(* Logix 5000 project; controller Hose_HP_Test_Rig_V1 vendor 1 type 14 code 149 rev 32.11; software revision 32.00; part 5 of 10 *)
(* tags used below, declared in another part *)
   CONS_ONS1 : BOOL;
   CONS_ONS2 : BOOL;
   CONS_ONS3 : BOOL;
   CONS_ONS4 : BOOL;
   DUMMY_VAL : REAL;
   EXHS_VAL_OFF_CE_STN1 : BOOL;
   EXHS_VAL_OFF_CE_STN2 : BOOL;
   EXHS_VAL_OFF_CE_STN3 : BOOL;
   FAULT_COMP_SENSOR : ALIAS FOR Local:2:I.Data.30;
   ONS42 : BOOL;
   ONS47 : BOOL;
   ONS48 : BOOL;
   ONS49 : BOOL;
   ONS53 : BOOL;
   ONS_74 : BOOL;
   ONS_75 : BOOL;
   ABORT_STN1 : BOOL;
   ABORT_STN2 : BOOL;
   ABORT_STN3 : BOOL;
   ABORT_STN4 : BOOL;
   AUTO_TEST_ON_STN1 : BOOL;
   AUTO_TEST_ON_STN2 : BOOL;
   AUTO_TEST_ON_STN3 : BOOL;
   AUTO_TEST_ON_STN4 : BOOL;
   BIN_MSG : DINT;
   BOTTOM_CLAMP_2BPR_HIGH : BOOL;
   BOTTOM_CLAMP_2BPR_LOW : BOOL;
   BOTTOM_CLAMP_4BPR_HIGH : BOOL;
   BOTTOM_CLAMP_4BPR_LOW : BOOL;
   BOTTOM_CLAMP_FAULT_STN1 : BOOL;
   BOTTOM_CLAMP_FAULT_STN2 : BOOL;
   BOTTOM_CLAMP_FAULT_STN3 : BOOL;
   BOTTOM_CLAMP_FAULT_STN4 : BOOL;
   BOTTOM_CLAMP_PR : REAL;
   BOTTOM_CLAMP_PR_DEL : TIMER;
   BOTTOM_CLAMP_PR_SEL : BOOL;
   BOTTOM_CLAMP_PR_SEQ : CLAMP_FAULT;
   BOTTOM_CLAMP_PS_STN2 : ALIAS FOR Local:2:I.Data.2;
   BOTTOM_CLAMP_PS_STN4 : ALIAS FOR Local:2:I.Data.12;
   BOTTOM_NOT_CLAMPED_STN1 : BOOL;
   CALB_START_PB_ONS_STN1 : BOOL;
   CALB_START_PB_ONS_STN2 : BOOL;
   CALB_START_PB_ONS_STN3 : BOOL;
   CALB_START_PB_ONS_STN4 : BOOL;
   CHECK_TRACE_STS_STN1 : BOOL;
   CLAMP_2BAR_HL : REAL;
   CLAMP_2BAR_LL : REAL;
   CLAMP_4BAR_HL : REAL;
   CLAMP_4BAR_LL : REAL;
   COMP_FAULT_STN1 : BOOL;
   CONS_CALB_ON_STN1 : BOOL;
   CONS_CALB_ON_STN2 : BOOL;
   CONS_CALB_ON_STN3 : BOOL;
   CONS_CALB_ON_STN4 : BOOL;
   CONS_CALB_TARRED_STN1 : BOOL;
   CONS_CALB_TARRED_STN2 : BOOL;
   CONS_CALB_TARRED_STN3 : BOOL;
   CONS_CALB_TARRED_STN4 : BOOL;
   CONS_DUMMIT_VAR : REAL;
   CONS_FILL_BLK_STN1 : CONSTRICTION_FILL_ON_SEQ;
   CONS_FILL_BLK_STN2 : CONSTRICTION_FILL_ON_SEQ;
   CONS_FILL_BLK_STN3 : CONSTRICTION_FILL_ON_SEQ;
   CONS_FILL_BLK_STN4 : CONSTRICTION_FILL_ON_SEQ;
   CONS_FILL_HIGH_STN1 : BOOL;
   CONS_FILL_HIGH_STN2 : BOOL;
   CONS_FILL_HIGH_STN3 : BOOL;
   CONS_FILL_HIGH_STN4 : BOOL;
   CONS_FILL_HL : REAL;
   CONS_FILL_LL : REAL;
   CONS_FILL_LOW_STN1 : BOOL;
   CONS_FILL_LOW_STN2 : BOOL;
   CONS_FILL_LOW_STN3 : BOOL;
   CONS_FILL_LOW_STN4 : BOOL;
   CONS_FILL_OFF_BLK_STN1 : CONSTRICTION_FILL_OFF_SEQ;
   CONS_FILL_OFF_BLK_STN2 : CONSTRICTION_FILL_OFF_SEQ;
   CONS_FILL_OFF_BLK_STN3 : CONSTRICTION_FILL_OFF_SEQ;
   CONS_FILL_OFF_BLK_STN4 : CONSTRICTION_FILL_OFF_SEQ;
   CONS_P2_STN1 : REAL;
   CONS_P2_STN2 : REAL;
   CONS_P2_STN3 : REAL;
   CONS_PR_BLK_STN1 : PR_CHECK;
   CONS_PR_BLK_STN2 : PR_CHECK;
   CONS_PR_BLK_STN3 : PR_CHECK;
   CONS_PR_BLK_STN4 : PR_CHECK;
   CONS_PR_P1_STN1 : REAL;
   CONS_PR_P1_STN2 : REAL;
   CONS_PR_P1_STN3 : REAL;
   CONS_PR_P1_STN4 : REAL;
   CONS_STS_STN1 : DINT;
   CONS_STS_STN2 : DINT;
   CONS_STS_STN3 : DINT;
   CONS_STS_STN4 : DINT;
   CONS_TEST_TIME_ACT : REAL;
   CONS_TEST_TIME_ACT_STN2 : REAL;
   CONS_TEST_TIME_ACT_STN3 : REAL;
   CONS_TEST_TIME_ACT_STN4 : REAL;
   CONS_TEST_TIME_SET : REAL;
   CONSTRICTION_BLK_STN1 : DROP_CHECK;
   CONSTRICTION_BLK_STN2 : DROP_CHECK;
   CONSTRICTION_BLK_STN3 : DROP_CHECK;
   CONSTRICTION_BLK_STN4 : DROP_CHECK;
   CONSTRICTION_FILL_OFF_STN1 : BOOL;
   CONSTRICTION_FILL_OFF_STN2 : BOOL;
   CONSTRICTION_FILL_OFF_STN3 : BOOL;
   CONSTRICTION_FILL_OFF_STN4 : BOOL;
   CONSTRICTION_FILL_VAL_STN1 : BOOL;
   CONSTRICTION_FILL_VAL_STN2 : BOOL;
   CONSTRICTION_FILL_VAL_STN3 : BOOL;
   CONSTRICTION_FILL_VAL_STN4 : BOOL;
   CONSTRICTION_NOK_STN1 : BOOL;
   CONSTRICTION_NOK_STN2 : BOOL;
   CONSTRICTION_NOK_STN3 : BOOL;
   CONSTRICTION_NOK_STN4 : BOOL;
   CONSTRICTION_OK_STN1 : BOOL;
   CONSTRICTION_OK_STN2 : BOOL;
   CONSTRICTION_OK_STN3 : BOOL;
   CONSTRICTION_OK_STN4 : BOOL;
   CONSTRICTION_TEST_ON_STN1 : BOOL;
   CONSTRICTION_TEST_ON_STN2 : BOOL;
   CONSTRICTION_TEST_ON_STN3 : BOOL;
   CONSTRICTION_TEST_ON_STN4 : BOOL;
   CYCLE_START_PB_STN1 : ALIAS FOR Local:1:I.Data.2;
   DOOR_CLOSE_ABORT_STN1 : BOOL;
   DOOR_NOT_CLOSED : BOOL;
   DOOR_NOT_OPEN_STN1 : BOOL;
   DROP_NOK_STN1 : BOOL;
   EC_STN1 : DINT;
   EC_STN2 : DINT;
   EC_STN3 : DINT;
   EC_STN4 : DINT;
   EMG_FAULT_CLR : BOOL;
   EMG_FAULTED_STN1 : BOOL;
   EMG_START_PB : ALIAS FOR Local:1:I.Data.6;
   EMG_STOP_PB_LH : ALIAS FOR Local:2:I.Data.23;
   EXHS_VAL_OFF_CE_STN4 : BOOL;
   EXHS_VAL_OFF_STN1 : BOOL;
   EXHS_VAL_OFF_STN2 : BOOL;
   EXHS_VAL_OFF_STN3 : BOOL;
   EXHS_VAL_OFF_STN4 : BOOL;
   EXHS_VAL_ON_STN1 : BOOL;
   EXHS_VAL_ON_STN2 : BOOL;
   EXHS_VAL_ON_STN3 : BOOL;
   EXHS_VAL_ON_STN4 : BOOL;
   FAIL_BIN_LOCK_PS : ALIAS FOR Local:2:I.Data.26;
   FAIL_CLR_ONS_STN1 : BOOL;
   FAIL_CLR_ONS_STN2 : BOOL;
   FAIL_CLR_ONS_STN3 : BOOL;
   FAIL_CLR_ONS_STN4 : BOOL;
   FAILED_STN1 : BOOL;
   FAILED_STN2 : BOOL;
   FAILED_STN3 : BOOL;
   FAULT_COUNT_STN1 : DINT;
   FAULT_COUNTER_STN1 : COUNTER;
   FAULTED_STN1 : BOOL;
   FAULTED_STN2 : BOOL;
   FAULTED_STN3 : BOOL;
   FAULTED_STN4 : BOOL;
   FILL_HIGH_STN1 : BOOL;
   FILL_LOW_STN1 : BOOL;
   FLT_CLR_ONS : BOOL;
   FLT_CLR_ONS_STN1 : BOOL;
   FLT_CLR_ONS_STN2 : BOOL;
   FLT_CLR_ONS_STN3 : BOOL;
   FLT_CLR_ONS_STN4 : BOOL;
   GOTO_FAULT_BIN_STN1 : DINT;
   HOME_COND_NOK_STN1 : BOOL;
   HOME_COND_OK_STN1 : BOOL;
   INIT_STN1 : BOOL;
   INIT_STN2 : BOOL;
   INIT_STN3 : BOOL;
   INIT_STN4 : BOOL;
   INLET_AIR_DPS : ALIAS FOR Local:1:I.Data.0;
   INLET_AIR_HPS : ALIAS FOR Local:1:I.Data.1;
   INLET_AIR_LOW : TIMER;
   INLET_AIR_SOL : ALIAS FOR Local:1:O.Data.0;
   LH_START_PB_STN2 : ALIAS FOR Local:1:I.Data.3;
   LH_START_PB_STN3 : ALIAS FOR Local:1:I.Data.4;
   LH_START_PB_STN4 : ALIAS FOR Local:1:I.Data.5;
   MSG_STN1 : DINT;
   MSG_STN2 : DINT;
   MSG_STN3 : DINT;
   MSG_STN4 : DINT;
   NO_COMP_FAULT_STN1 : BOOL;
   NO_SYSTEM_FAULT_STN1 : BOOL;
   NOT_FAILED_STN1 : BOOL;
   PASS_BIN_FULL : DINT;
   PR_DIFF_ACT_STN1 : REAL;
   PR_DIFF_ACT_STN2 : REAL;
   PR_DIFF_ACT_STN3 : REAL;
   PR_DIFF_ACT_STN4 : REAL;
   PR_DIFF_CALB_ACT : REAL;
   PR_DIFF_HL : REAL;
   PR_DIFF_LL : REAL;
   PR_DIFF_TARRED_STN1 : REAL;
   PR_DIFF_TARRED_STN2 : REAL;
   PR_DIFF_TARRED_STN3 : REAL;
   PR_DIFF_TARRED_STN4 : REAL;
   RETEST : BOOL;
   RST_DOOR_NOT_OPEN_STN1 : BOOL;
   RST_EXHS_VAL_OFF_STN1 : BOOL;
   RST_EXHS_VAL_OFF_STN2 : BOOL;
   RST_EXHS_VAL_OFF_STN3 : BOOL;
   RST_EXHS_VAL_OFF_STN4 : BOOL;
   RST_SEQ_ON_STN1 : BOOL;
   RST_SEQ_ON_STN2 : BOOL;
   RST_SEQ_ON_STN3 : BOOL;
   RST_SEQ_ON_STN4 : BOOL;
   SCR_STS : DINT[6];
   SEQ_NO_STN1 : DINT;
   SEQ_NO_STN2 : DINT;
   SEQ_NO_STN3 : DINT;
   SEQ_NO_STN4 : DINT;
   STAB_HIGH_STN1 : BOOL;
   STAB_LOW_STN1 : BOOL;
   STAMP_HL : REAL;
   STAMP_LL : REAL;
   STAMP_NOT_FWD : BOOL;
   STAMP_NOT_RET : BOOL;
   STAMP_PR : REAL;
   STAMP_PR_CHECK : TIMER;
   STAMP_PR_DEL : TIMER;
   STAMP_PR_HIGH_STN1 : BOOL;
   STAMP_PR_LOW_STN1 : BOOL;
   STAMP_SOL_STN1 : ALIAS FOR Local:1:O.Data.5;
   STS : DINT;
   SYSTEM_FAULT_STN1 : BOOL;
   TARRED_VALUE_STN1 : REAL;
   TARRED_VALUE_STN2 : REAL;
   TARRED_VALUE_STN3 : REAL;
   TARRED_VALUE_STN4 : REAL;
   TEST_ON_STN1 : BOOL;
   TEST_ON_STN2 : BOOL;
   TEST_ON_STN3 : BOOL;
   TEST_ON_STN4 : BOOL;
   TEST_STS_STN1 : DINT;
   TEST_STS_STN2 : DINT;
   TEST_STS_STN3 : DINT;
   TEST_STS_STN4 : DINT;
   TOP_CLAMP_2BPR_HIGH : BOOL;
   TOP_CLAMP_2BPR_LOW : BOOL;
   TOP_CLAMP_4BPR_HIGH : BOOL;
   TOP_CLAMP_4BPR_LOW : BOOL;
   TOP_CLAMP_FAULT_STN1 : BOOL;
   TOP_CLAMP_FAULT_STN2 : BOOL;
   TOP_CLAMP_FAULT_STN3 : BOOL;
   TOP_CLAMP_FAULT_STN4 : BOOL;
   TOP_CLAMP_PR : REAL;
   TOP_CLAMP_PR_CHK_STN1 : TIMER;
   TOP_CLAMP_PR_DEL : TIMER;
   TOP_CLAMP_PR_SEL : BOOL;
(* MainProgram, continued *)

ROUTINE Constriction_Stn1   (* ladder *)
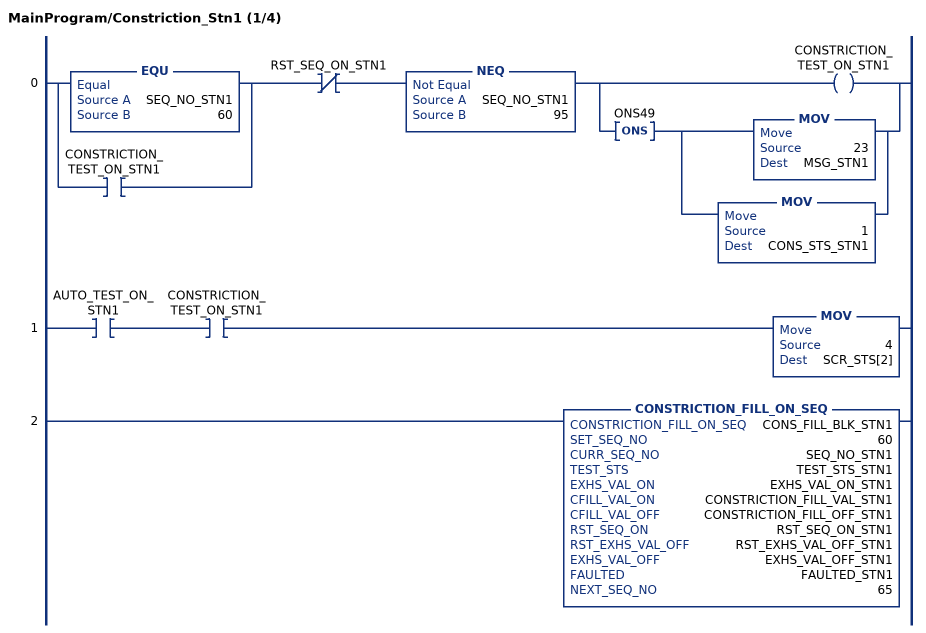
   0: [EQU(SEQ_NO_STN1,60) ,XIC(CONSTRICTION_TEST_ON_STN1) ]XIO(RST_SEQ_ON_STN1)NEQ(SEQ_NO_STN1,95)[OTE(CONSTRICTION_TEST_ON_STN1) ,ONS(ONS49) [MOV(23,MSG_STN1) ,MOV(1,CONS_STS_STN1) ] ];
   1: XIC(AUTO_TEST_ON_STN1)XIC(CONSTRICTION_TEST_ON_STN1)MOV(4,SCR_STS[2]);
   2: CONSTRICTION_FILL_ON_SEQ(CONS_FILL_BLK_STN1,60,SEQ_NO_STN1,TEST_STS_STN1,EXHS_VAL_ON_STN1,CONSTRICTION_FILL_VAL_STN1,CONSTRICTION_FILL_OFF_STN1,RST_SEQ_ON_STN1,RST_EXHS_VAL_OFF_STN1,EXHS_VAL_OFF_STN1,FAULTED_STN1,65);
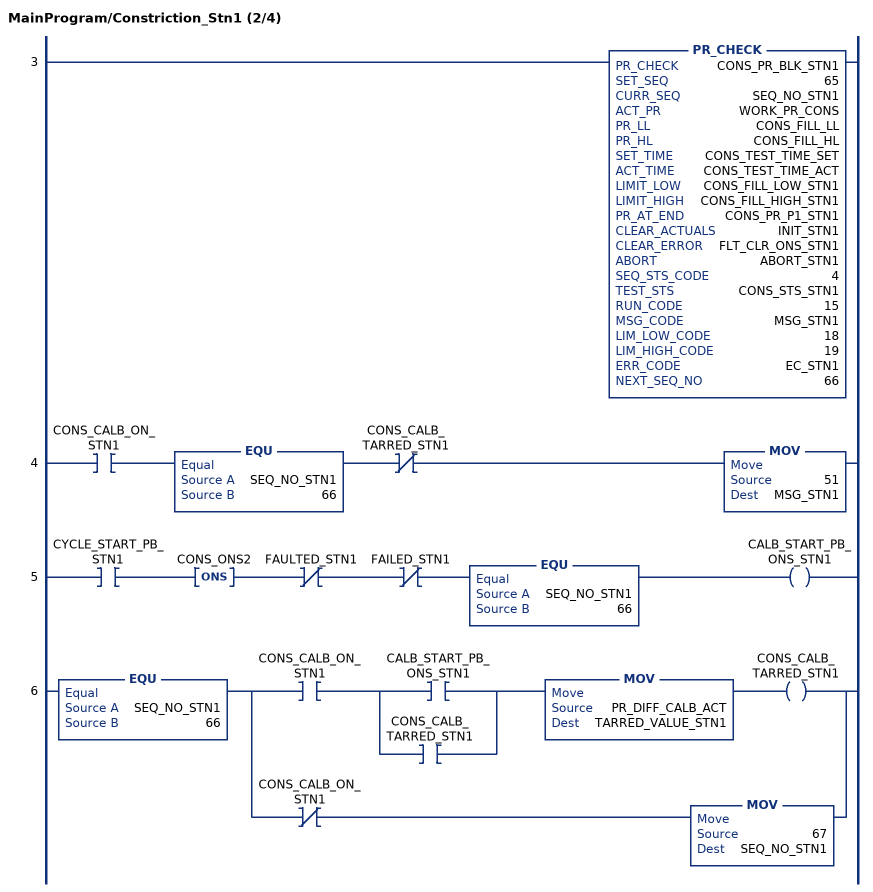
   3: PR_CHECK(CONS_PR_BLK_STN1,65,SEQ_NO_STN1,WORK_PR_CONS,CONS_FILL_LL,CONS_FILL_HL,CONS_TEST_TIME_SET,CONS_TEST_TIME_ACT,CONS_FILL_LOW_STN1,CONS_FILL_HIGH_STN1,CONS_PR_P1_STN1,INIT_STN1,FLT_CLR_ONS_STN1,ABORT_STN1,4,CONS_STS_STN1,15,MSG_STN1,18,19,EC_STN1,66);
   4: XIC(CONS_CALB_ON_STN1)EQU(SEQ_NO_STN1,66)XIO(CONS_CALB_TARRED_STN1)MOV(51,MSG_STN1);
   5: XIC(CYCLE_START_PB_STN1)ONS(CONS_ONS2)XIO(FAULTED_STN1)XIO(FAILED_STN1)EQU(SEQ_NO_STN1,66)OTE(CALB_START_PB_ONS_STN1);
   6: EQU(SEQ_NO_STN1,66)[XIC(CONS_CALB_ON_STN1) [XIC(CALB_START_PB_ONS_STN1) ,XIC(CONS_CALB_TARRED_STN1) ] MOV(PR_DIFF_CALB_ACT,TARRED_VALUE_STN1) OTE(CONS_CALB_TARRED_STN1) ,XIO(CONS_CALB_ON_STN1) MOV(67,SEQ_NO_STN1) ];
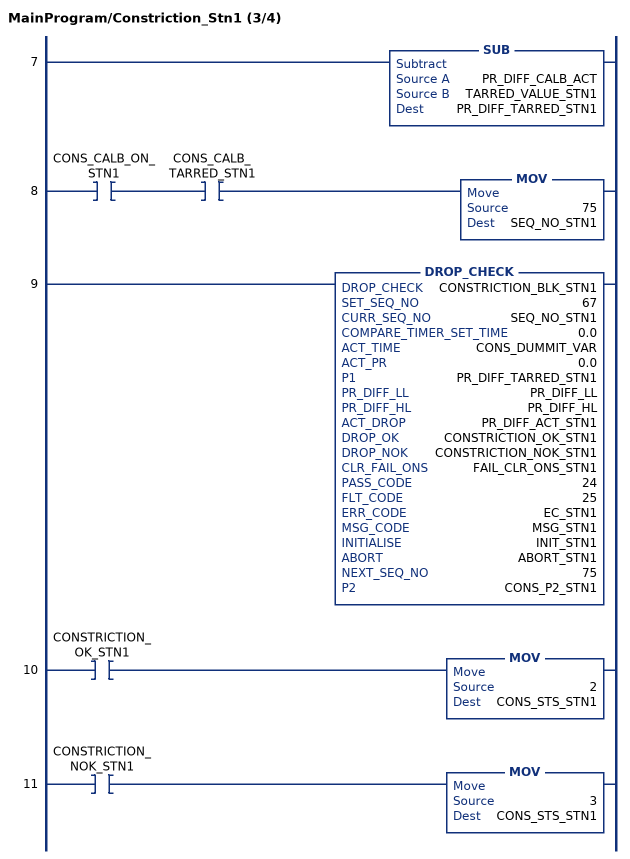
   7: SUB(PR_DIFF_CALB_ACT,TARRED_VALUE_STN1,PR_DIFF_TARRED_STN1);
   8: XIC(CONS_CALB_ON_STN1)XIC(CONS_CALB_TARRED_STN1)MOV(75,SEQ_NO_STN1);
   9: DROP_CHECK(CONSTRICTION_BLK_STN1,67,SEQ_NO_STN1,0.0,CONS_DUMMIT_VAR,0.0,PR_DIFF_TARRED_STN1,PR_DIFF_LL,PR_DIFF_HL,PR_DIFF_ACT_STN1,CONSTRICTION_OK_STN1,CONSTRICTION_NOK_STN1,FAIL_CLR_ONS_STN1,24,25,EC_STN1,MSG_STN1,INIT_STN1,ABORT_STN1,75,CONS_P2_STN1);
   10: XIC(CONSTRICTION_OK_STN1)MOV(2,CONS_STS_STN1);
   11: XIC(CONSTRICTION_NOK_STN1)MOV(3,CONS_STS_STN1);
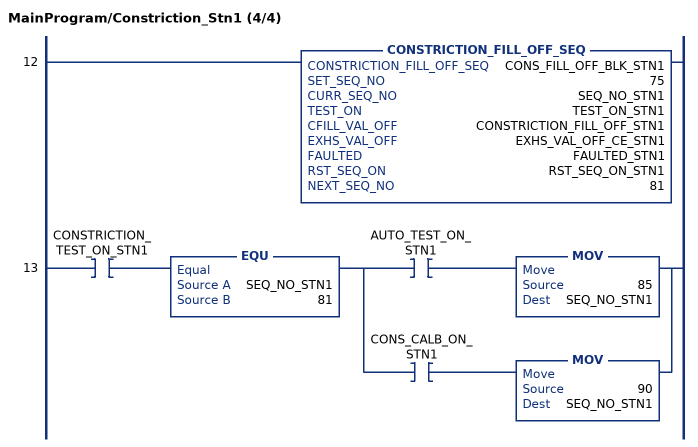
   12: CONSTRICTION_FILL_OFF_SEQ(CONS_FILL_OFF_BLK_STN1,75,SEQ_NO_STN1,TEST_ON_STN1,CONSTRICTION_FILL_OFF_STN1,EXHS_VAL_OFF_CE_STN1,FAULTED_STN1,RST_SEQ_ON_STN1,81);
   13: XIC(CONSTRICTION_TEST_ON_STN1)EQU(SEQ_NO_STN1,81)[XIC(AUTO_TEST_ON_STN1) MOV(85,SEQ_NO_STN1) ,XIC(CONS_CALB_ON_STN1) MOV(90,SEQ_NO_STN1) ];
END_ROUTINE

ROUTINE Constriction_Stn2   (* ladder *)
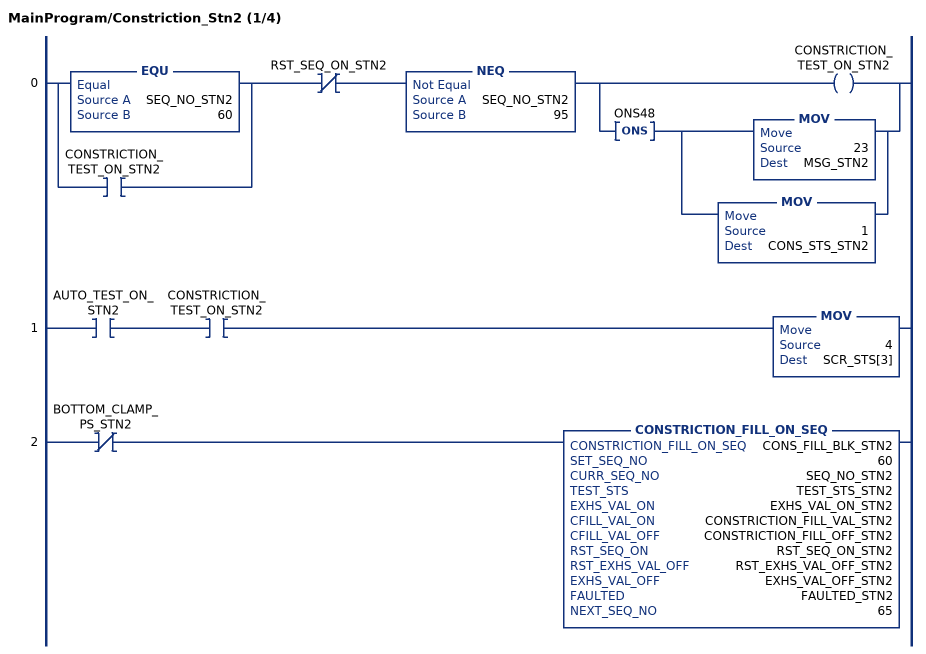
   0: [EQU(SEQ_NO_STN2,60) ,XIC(CONSTRICTION_TEST_ON_STN2) ]XIO(RST_SEQ_ON_STN2)NEQ(SEQ_NO_STN2,95)[OTE(CONSTRICTION_TEST_ON_STN2) ,ONS(ONS48) [MOV(23,MSG_STN2) ,MOV(1,CONS_STS_STN2) ] ];
   1: XIC(AUTO_TEST_ON_STN2)XIC(CONSTRICTION_TEST_ON_STN2)MOV(4,SCR_STS[3]);
   2: XIO(BOTTOM_CLAMP_PS_STN2)CONSTRICTION_FILL_ON_SEQ(CONS_FILL_BLK_STN2,60,SEQ_NO_STN2,TEST_STS_STN2,EXHS_VAL_ON_STN2,CONSTRICTION_FILL_VAL_STN2,CONSTRICTION_FILL_OFF_STN2,RST_SEQ_ON_STN2,RST_EXHS_VAL_OFF_STN2,EXHS_VAL_OFF_STN2,FAULTED_STN2,65);
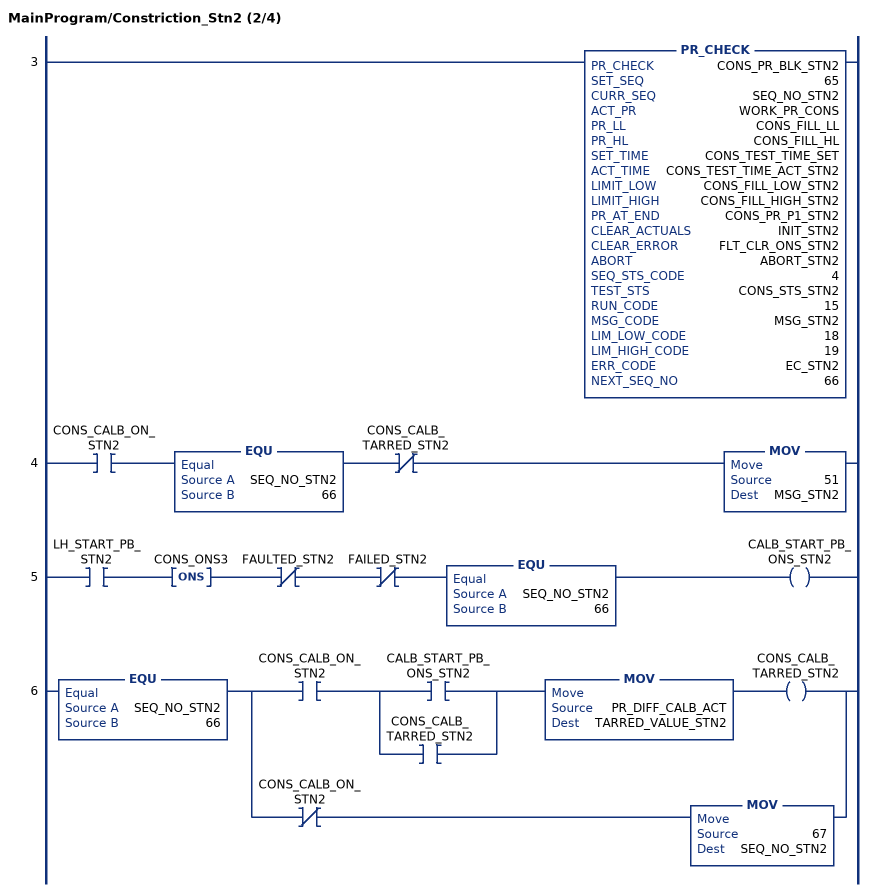
   3: PR_CHECK(CONS_PR_BLK_STN2,65,SEQ_NO_STN2,WORK_PR_CONS,CONS_FILL_LL,CONS_FILL_HL,CONS_TEST_TIME_SET,CONS_TEST_TIME_ACT_STN2,CONS_FILL_LOW_STN2,CONS_FILL_HIGH_STN2,CONS_PR_P1_STN2,INIT_STN2,FLT_CLR_ONS_STN2,ABORT_STN2,4,CONS_STS_STN2,15,MSG_STN2,18,19,EC_STN2,66);
   4: XIC(CONS_CALB_ON_STN2)EQU(SEQ_NO_STN2,66)XIO(CONS_CALB_TARRED_STN2)MOV(51,MSG_STN2);
   5: XIC(LH_START_PB_STN2)ONS(CONS_ONS3)XIO(FAULTED_STN2)XIO(FAILED_STN2)EQU(SEQ_NO_STN2,66)OTE(CALB_START_PB_ONS_STN2);
   6: EQU(SEQ_NO_STN2,66)[XIC(CONS_CALB_ON_STN2) [XIC(CALB_START_PB_ONS_STN2) ,XIC(CONS_CALB_TARRED_STN2) ] MOV(PR_DIFF_CALB_ACT,TARRED_VALUE_STN2) OTE(CONS_CALB_TARRED_STN2) ,XIO(CONS_CALB_ON_STN2) MOV(67,SEQ_NO_STN2) ];
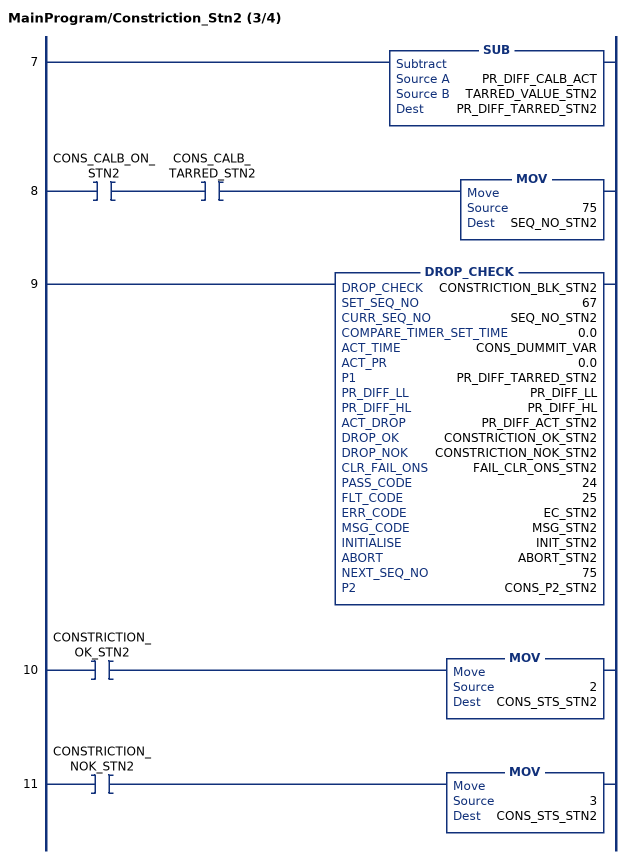
   7: SUB(PR_DIFF_CALB_ACT,TARRED_VALUE_STN2,PR_DIFF_TARRED_STN2);
   8: XIC(CONS_CALB_ON_STN2)XIC(CONS_CALB_TARRED_STN2)MOV(75,SEQ_NO_STN2);
   9: DROP_CHECK(CONSTRICTION_BLK_STN2,67,SEQ_NO_STN2,0.0,CONS_DUMMIT_VAR,0.0,PR_DIFF_TARRED_STN2,PR_DIFF_LL,PR_DIFF_HL,PR_DIFF_ACT_STN2,CONSTRICTION_OK_STN2,CONSTRICTION_NOK_STN2,FAIL_CLR_ONS_STN2,24,25,EC_STN2,MSG_STN2,INIT_STN2,ABORT_STN2,75,CONS_P2_STN2);
   10: XIC(CONSTRICTION_OK_STN2)MOV(2,CONS_STS_STN2);
   11: XIC(CONSTRICTION_NOK_STN2)MOV(3,CONS_STS_STN2);
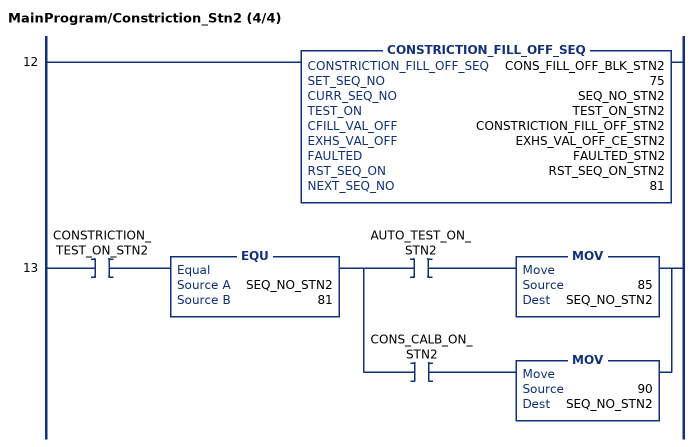
   12: CONSTRICTION_FILL_OFF_SEQ(CONS_FILL_OFF_BLK_STN2,75,SEQ_NO_STN2,TEST_ON_STN2,CONSTRICTION_FILL_OFF_STN2,EXHS_VAL_OFF_CE_STN2,FAULTED_STN2,RST_SEQ_ON_STN2,81);
   13: XIC(CONSTRICTION_TEST_ON_STN2)EQU(SEQ_NO_STN2,81)[XIC(AUTO_TEST_ON_STN2) MOV(85,SEQ_NO_STN2) ,XIC(CONS_CALB_ON_STN2) MOV(90,SEQ_NO_STN2) ];
END_ROUTINE

ROUTINE Constriction_Stn3   (* ladder *)
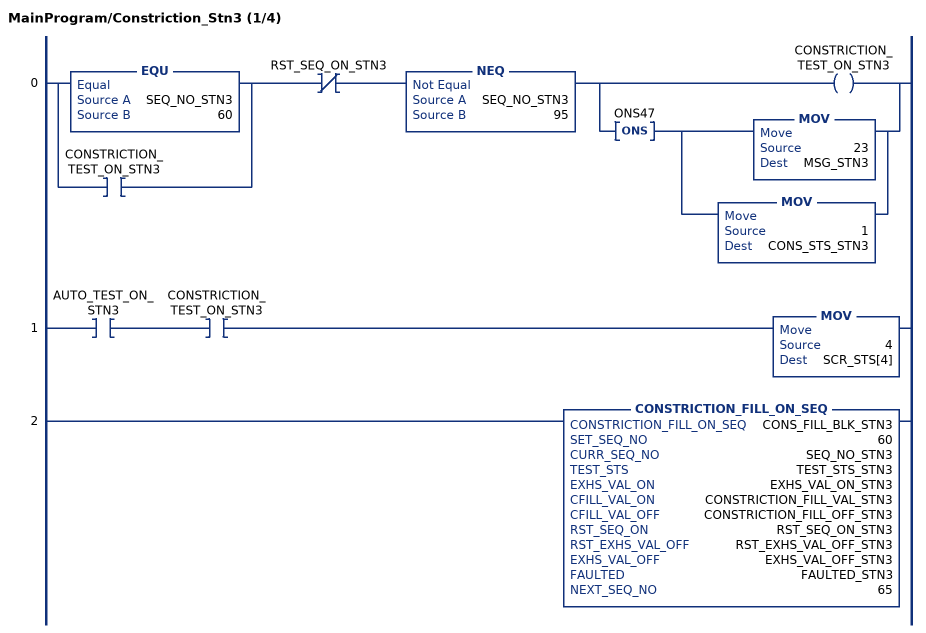
   0: [EQU(SEQ_NO_STN3,60) ,XIC(CONSTRICTION_TEST_ON_STN3) ]XIO(RST_SEQ_ON_STN3)NEQ(SEQ_NO_STN3,95)[OTE(CONSTRICTION_TEST_ON_STN3) ,ONS(ONS47) [MOV(23,MSG_STN3) ,MOV(1,CONS_STS_STN3) ] ];
   1: XIC(AUTO_TEST_ON_STN3)XIC(CONSTRICTION_TEST_ON_STN3)MOV(4,SCR_STS[4]);
   2: CONSTRICTION_FILL_ON_SEQ(CONS_FILL_BLK_STN3,60,SEQ_NO_STN3,TEST_STS_STN3,EXHS_VAL_ON_STN3,CONSTRICTION_FILL_VAL_STN3,CONSTRICTION_FILL_OFF_STN3,RST_SEQ_ON_STN3,RST_EXHS_VAL_OFF_STN3,EXHS_VAL_OFF_STN3,FAULTED_STN3,65);
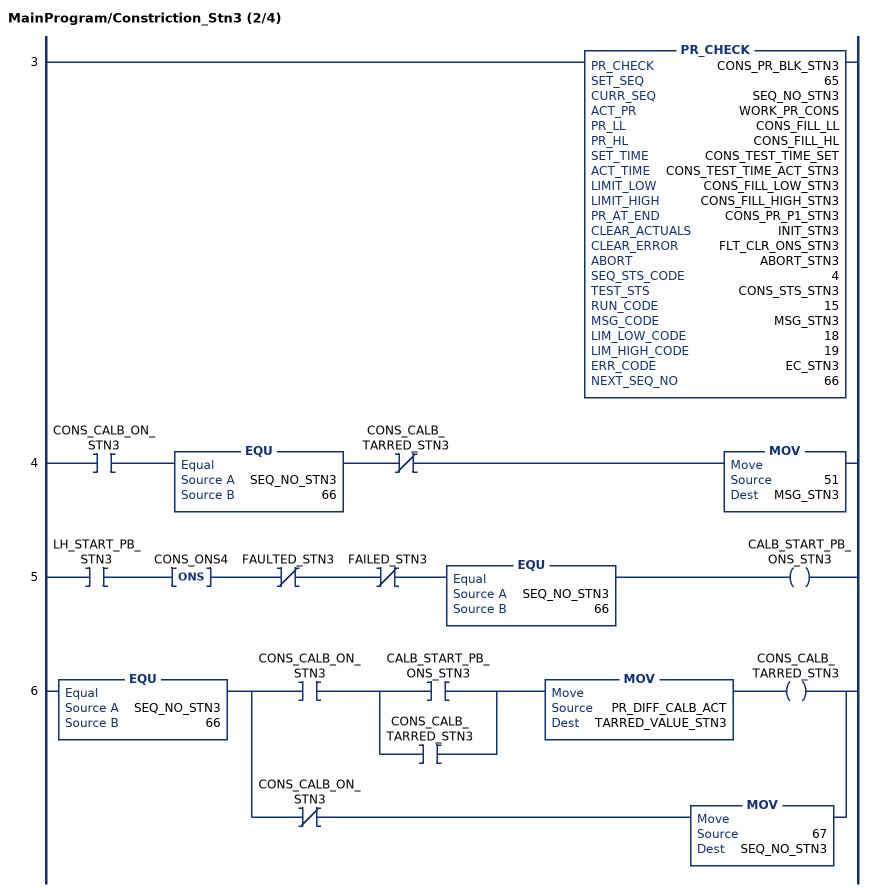
   3: PR_CHECK(CONS_PR_BLK_STN3,65,SEQ_NO_STN3,WORK_PR_CONS,CONS_FILL_LL,CONS_FILL_HL,CONS_TEST_TIME_SET,CONS_TEST_TIME_ACT_STN3,CONS_FILL_LOW_STN3,CONS_FILL_HIGH_STN3,CONS_PR_P1_STN3,INIT_STN3,FLT_CLR_ONS_STN3,ABORT_STN3,4,CONS_STS_STN3,15,MSG_STN3,18,19,EC_STN3,66);
   4: XIC(CONS_CALB_ON_STN3)EQU(SEQ_NO_STN3,66)XIO(CONS_CALB_TARRED_STN3)MOV(51,MSG_STN3);
   5: XIC(LH_START_PB_STN3)ONS(CONS_ONS4)XIO(FAULTED_STN3)XIO(FAILED_STN3)EQU(SEQ_NO_STN3,66)OTE(CALB_START_PB_ONS_STN3);
   6: EQU(SEQ_NO_STN3,66)[XIC(CONS_CALB_ON_STN3) [XIC(CALB_START_PB_ONS_STN3) ,XIC(CONS_CALB_TARRED_STN3) ] MOV(PR_DIFF_CALB_ACT,TARRED_VALUE_STN3) OTE(CONS_CALB_TARRED_STN3) ,XIO(CONS_CALB_ON_STN3) MOV(67,SEQ_NO_STN3) ];
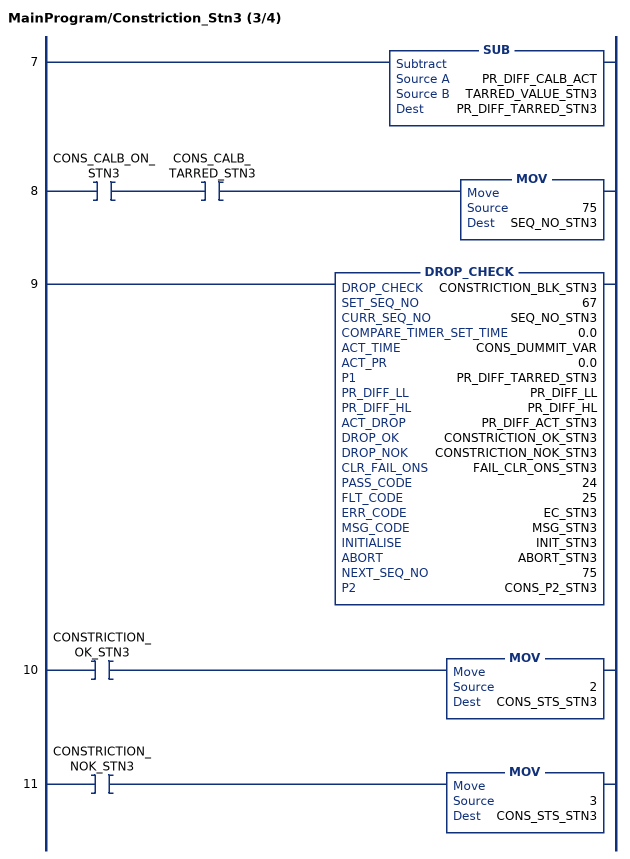
   7: SUB(PR_DIFF_CALB_ACT,TARRED_VALUE_STN3,PR_DIFF_TARRED_STN3);
   8: XIC(CONS_CALB_ON_STN3)XIC(CONS_CALB_TARRED_STN3)MOV(75,SEQ_NO_STN3);
   9: DROP_CHECK(CONSTRICTION_BLK_STN3,67,SEQ_NO_STN3,0.0,CONS_DUMMIT_VAR,0.0,PR_DIFF_TARRED_STN3,PR_DIFF_LL,PR_DIFF_HL,PR_DIFF_ACT_STN3,CONSTRICTION_OK_STN3,CONSTRICTION_NOK_STN3,FAIL_CLR_ONS_STN3,24,25,EC_STN3,MSG_STN3,INIT_STN3,ABORT_STN3,75,CONS_P2_STN3);
   10: XIC(CONSTRICTION_OK_STN3)MOV(2,CONS_STS_STN3);
   11: XIC(CONSTRICTION_NOK_STN3)MOV(3,CONS_STS_STN3);
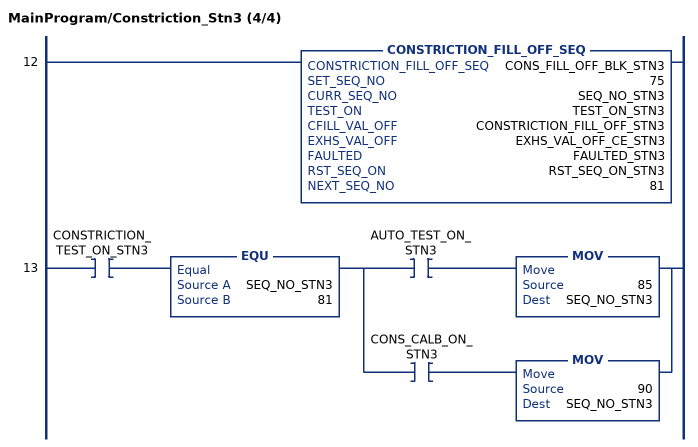
   12: CONSTRICTION_FILL_OFF_SEQ(CONS_FILL_OFF_BLK_STN3,75,SEQ_NO_STN3,TEST_ON_STN3,CONSTRICTION_FILL_OFF_STN3,EXHS_VAL_OFF_CE_STN3,FAULTED_STN3,RST_SEQ_ON_STN3,81);
   13: XIC(CONSTRICTION_TEST_ON_STN3)EQU(SEQ_NO_STN3,81)[XIC(AUTO_TEST_ON_STN3) MOV(85,SEQ_NO_STN3) ,XIC(CONS_CALB_ON_STN3) MOV(90,SEQ_NO_STN3) ];
END_ROUTINE

ROUTINE Constriction_Stn4   (* ladder *)
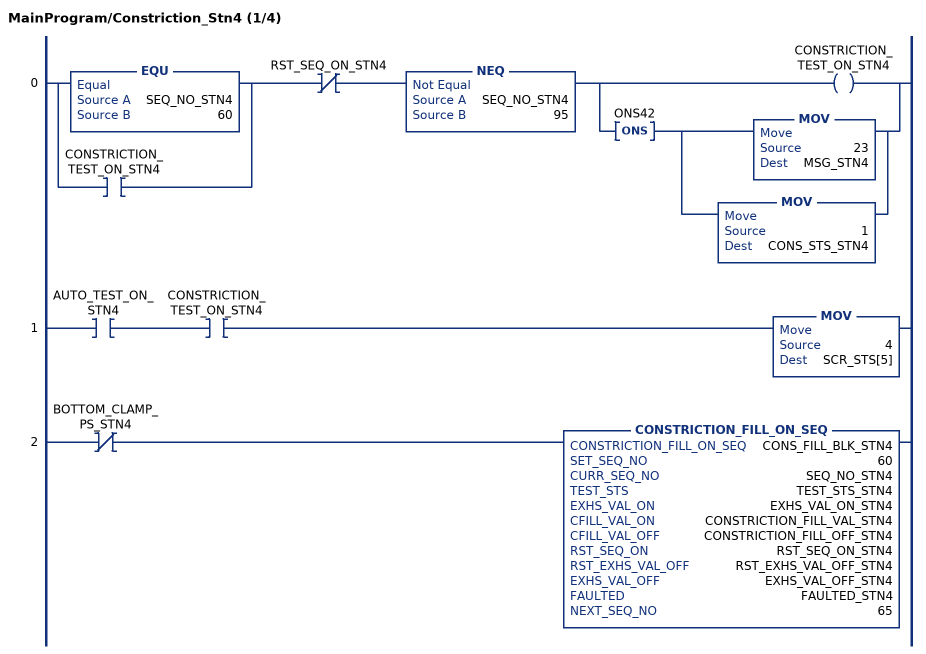
   0: [EQU(SEQ_NO_STN4,60) ,XIC(CONSTRICTION_TEST_ON_STN4) ]XIO(RST_SEQ_ON_STN4)NEQ(SEQ_NO_STN4,95)[OTE(CONSTRICTION_TEST_ON_STN4) ,ONS(ONS42) [MOV(23,MSG_STN4) ,MOV(1,CONS_STS_STN4) ] ];
   1: XIC(AUTO_TEST_ON_STN4)XIC(CONSTRICTION_TEST_ON_STN4)MOV(4,SCR_STS[5]);
   2: XIO(BOTTOM_CLAMP_PS_STN4)CONSTRICTION_FILL_ON_SEQ(CONS_FILL_BLK_STN4,60,SEQ_NO_STN4,TEST_STS_STN4,EXHS_VAL_ON_STN4,CONSTRICTION_FILL_VAL_STN4,CONSTRICTION_FILL_OFF_STN4,RST_SEQ_ON_STN4,RST_EXHS_VAL_OFF_STN4,EXHS_VAL_OFF_STN4,FAULTED_STN4,65);
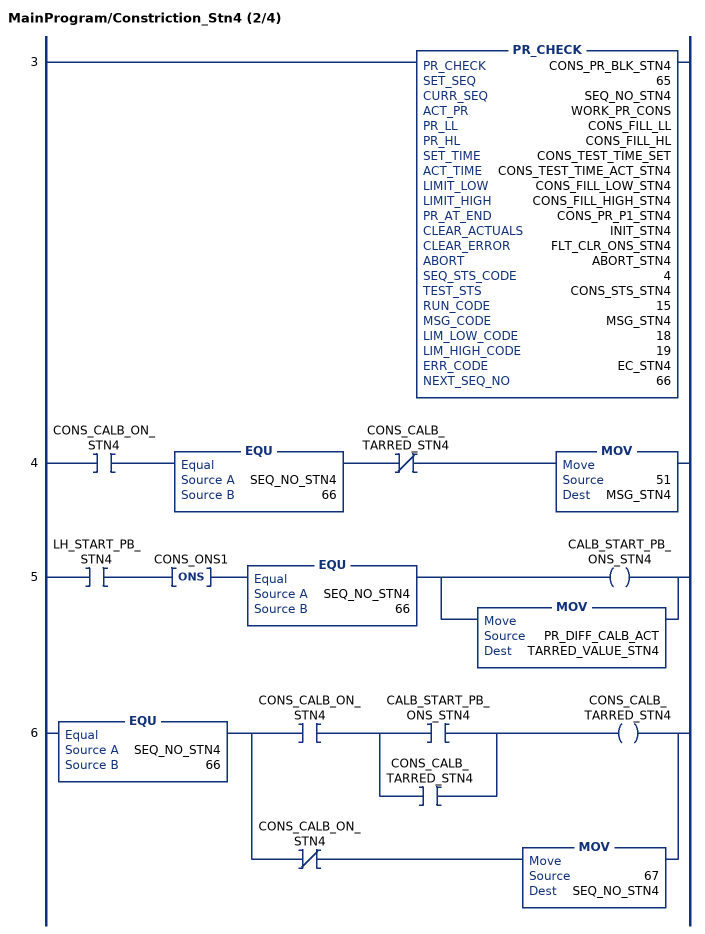
   3: PR_CHECK(CONS_PR_BLK_STN4,65,SEQ_NO_STN4,WORK_PR_CONS,CONS_FILL_LL,CONS_FILL_HL,CONS_TEST_TIME_SET,CONS_TEST_TIME_ACT_STN4,CONS_FILL_LOW_STN4,CONS_FILL_HIGH_STN4,CONS_PR_P1_STN4,INIT_STN4,FLT_CLR_ONS_STN4,ABORT_STN4,4,CONS_STS_STN4,15,MSG_STN4,18,19,EC_STN4,66);
   4: XIC(CONS_CALB_ON_STN4)EQU(SEQ_NO_STN4,66)XIO(CONS_CALB_TARRED_STN4)MOV(51,MSG_STN4);
   5: XIC(LH_START_PB_STN4)ONS(CONS_ONS1)EQU(SEQ_NO_STN4,66)[OTE(CALB_START_PB_ONS_STN4) ,MOV(PR_DIFF_CALB_ACT,TARRED_VALUE_STN4) ];
   6: EQU(SEQ_NO_STN4,66)[XIC(CONS_CALB_ON_STN4) [XIC(CALB_START_PB_ONS_STN4) ,XIC(CONS_CALB_TARRED_STN4) ] OTE(CONS_CALB_TARRED_STN4) ,XIO(CONS_CALB_ON_STN4) MOV(67,SEQ_NO_STN4) ];
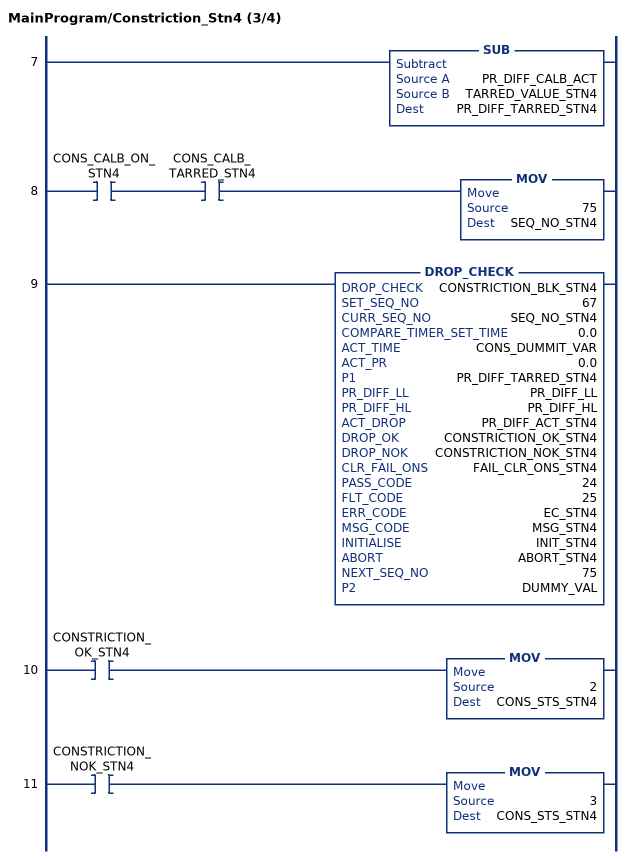
   7: SUB(PR_DIFF_CALB_ACT,TARRED_VALUE_STN4,PR_DIFF_TARRED_STN4);
   8: XIC(CONS_CALB_ON_STN4)XIC(CONS_CALB_TARRED_STN4)MOV(75,SEQ_NO_STN4);
   9: DROP_CHECK(CONSTRICTION_BLK_STN4,67,SEQ_NO_STN4,0.0,CONS_DUMMIT_VAR,0.0,PR_DIFF_TARRED_STN4,PR_DIFF_LL,PR_DIFF_HL,PR_DIFF_ACT_STN4,CONSTRICTION_OK_STN4,CONSTRICTION_NOK_STN4,FAIL_CLR_ONS_STN4,24,25,EC_STN4,MSG_STN4,INIT_STN4,ABORT_STN4,75,DUMMY_VAL);
   10: XIC(CONSTRICTION_OK_STN4)MOV(2,CONS_STS_STN4);
   11: XIC(CONSTRICTION_NOK_STN4)MOV(3,CONS_STS_STN4);
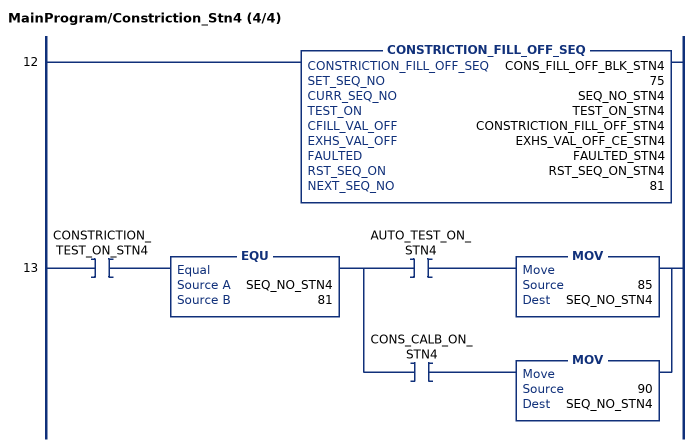
   12: CONSTRICTION_FILL_OFF_SEQ(CONS_FILL_OFF_BLK_STN4,75,SEQ_NO_STN4,TEST_ON_STN4,CONSTRICTION_FILL_OFF_STN4,EXHS_VAL_OFF_CE_STN4,FAULTED_STN4,RST_SEQ_ON_STN4,81);
   13: XIC(CONSTRICTION_TEST_ON_STN4)EQU(SEQ_NO_STN4,81)[XIC(AUTO_TEST_ON_STN4) MOV(85,SEQ_NO_STN4) ,XIC(CONS_CALB_ON_STN4) MOV(90,SEQ_NO_STN4) ];
END_ROUTINE

ROUTINE Fault_Fail_Msg   (* ladder *)
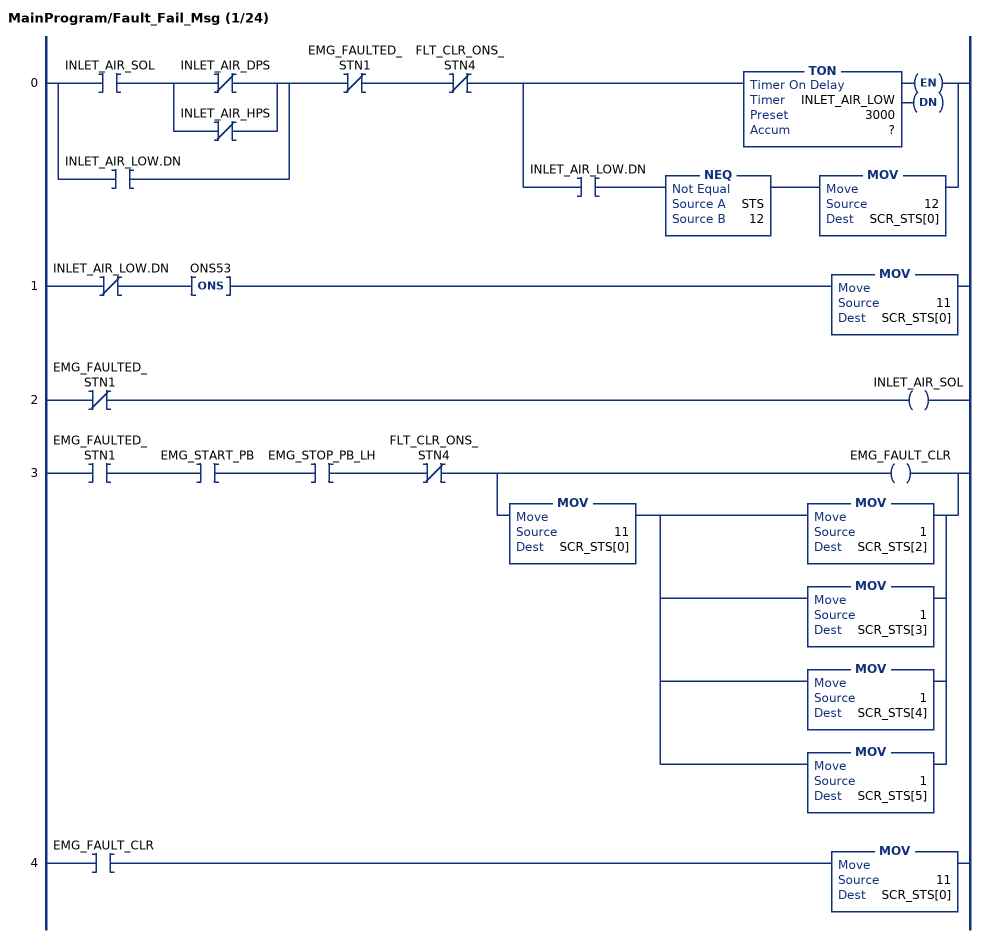
   0: [XIC(INLET_AIR_SOL) [XIO(INLET_AIR_DPS) ,XIO(INLET_AIR_HPS) ] ,XIC(INLET_AIR_LOW.DN) ]XIO(EMG_FAULTED_STN1)XIO(FLT_CLR_ONS_STN4)[TON(INLET_AIR_LOW,?,?) ,XIC(INLET_AIR_LOW.DN) NEQ(STS,12) MOV(12,SCR_STS[0]) ];
   1: XIO(INLET_AIR_LOW.DN)ONS(ONS53)MOV(11,SCR_STS[0]);
   2: XIO(EMG_FAULTED_STN1)OTE(INLET_AIR_SOL);
   3: XIC(EMG_FAULTED_STN1)XIC(EMG_START_PB)XIC(EMG_STOP_PB_LH)XIO(FLT_CLR_ONS_STN4)[OTE(EMG_FAULT_CLR) ,MOV(11,SCR_STS[0]) [MOV(1,SCR_STS[2]) ,MOV(1,SCR_STS[3]) ,MOV(1,SCR_STS[4]) ,MOV(1,SCR_STS[5]) ] ];
   4: XIC(EMG_FAULT_CLR)MOV(11,SCR_STS[0]);
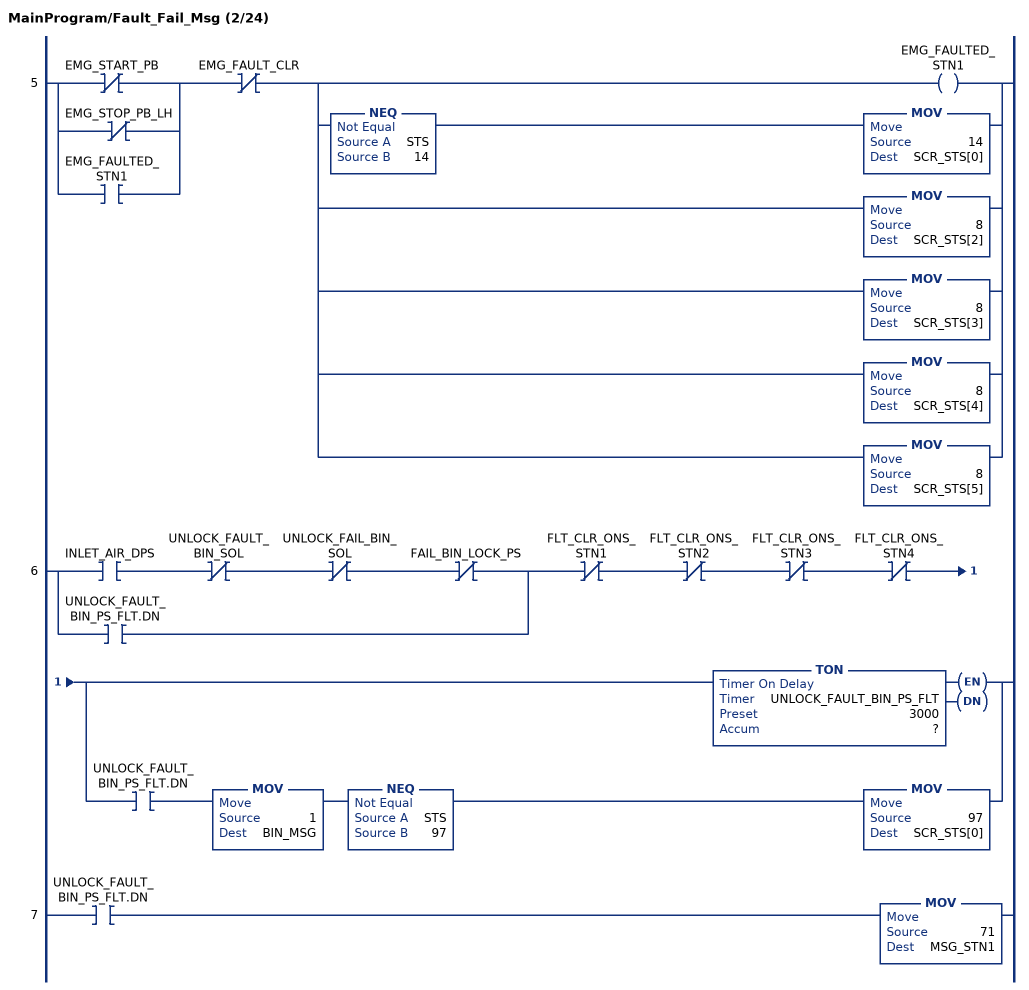
   5: [XIO(EMG_START_PB) ,XIO(EMG_STOP_PB_LH) ,XIC(EMG_FAULTED_STN1) ]XIO(EMG_FAULT_CLR)[OTE(EMG_FAULTED_STN1) ,NEQ(STS,14) MOV(14,SCR_STS[0]) ,MOV(8,SCR_STS[2]) ,MOV(8,SCR_STS[3]) ,MOV(8,SCR_STS[4]) ,MOV(8,SCR_STS[5]) ];
   6: [XIC(INLET_AIR_DPS) XIO(UNLOCK_FAULT_BIN_SOL) XIO(UNLOCK_FAIL_BIN_SOL) XIO(FAIL_BIN_LOCK_PS) ,XIC(UNLOCK_FAULT_BIN_PS_FLT.DN) ]XIO(FLT_CLR_ONS_STN1)XIO(FLT_CLR_ONS_STN2)XIO(FLT_CLR_ONS_STN3)XIO(FLT_CLR_ONS_STN4)[TON(UNLOCK_FAULT_BIN_PS_FLT,?,?) ,XIC(UNLOCK_FAULT_BIN_PS_FLT.DN) MOV(1,BIN_MSG) NEQ(STS,97) MOV(97,SCR_STS[0]) ];
   7: XIC(UNLOCK_FAULT_BIN_PS_FLT.DN)MOV(71,MSG_STN1);
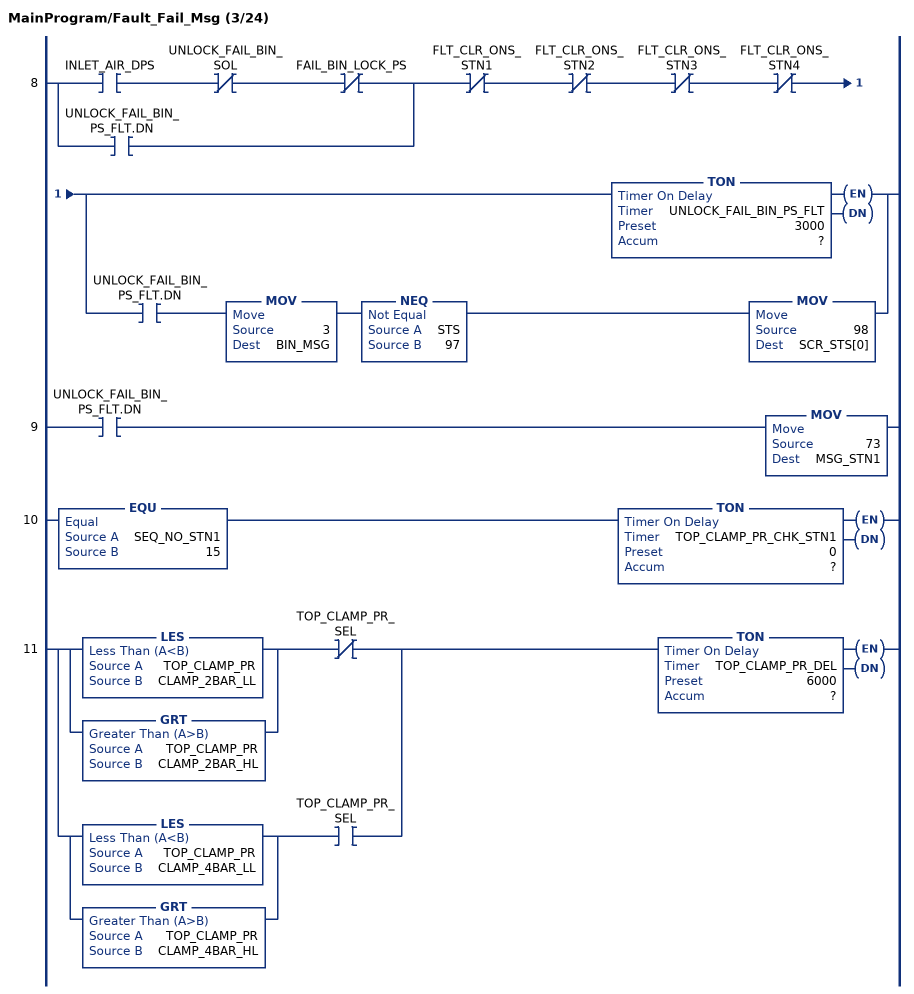
   8: [XIC(INLET_AIR_DPS) XIO(UNLOCK_FAIL_BIN_SOL) XIO(FAIL_BIN_LOCK_PS) ,XIC(UNLOCK_FAIL_BIN_PS_FLT.DN) ]XIO(FLT_CLR_ONS_STN1)XIO(FLT_CLR_ONS_STN2)XIO(FLT_CLR_ONS_STN3)XIO(FLT_CLR_ONS_STN4)[TON(UNLOCK_FAIL_BIN_PS_FLT,?,?) ,XIC(UNLOCK_FAIL_BIN_PS_FLT.DN) MOV(3,BIN_MSG) NEQ(STS,97) MOV(98,SCR_STS[0]) ];
   9: XIC(UNLOCK_FAIL_BIN_PS_FLT.DN)MOV(73,MSG_STN1);
   10: EQU(SEQ_NO_STN1,15)TON(TOP_CLAMP_PR_CHK_STN1,?,?);
   11: [[LES(TOP_CLAMP_PR,CLAMP_2BAR_LL) ,GRT(TOP_CLAMP_PR,CLAMP_2BAR_HL) ] XIO(TOP_CLAMP_PR_SEL) ,[LES(TOP_CLAMP_PR,CLAMP_4BAR_LL) ,GRT(TOP_CLAMP_PR,CLAMP_4BAR_HL) ] XIC(TOP_CLAMP_PR_SEL) ]TON(TOP_CLAMP_PR_DEL,?,?);
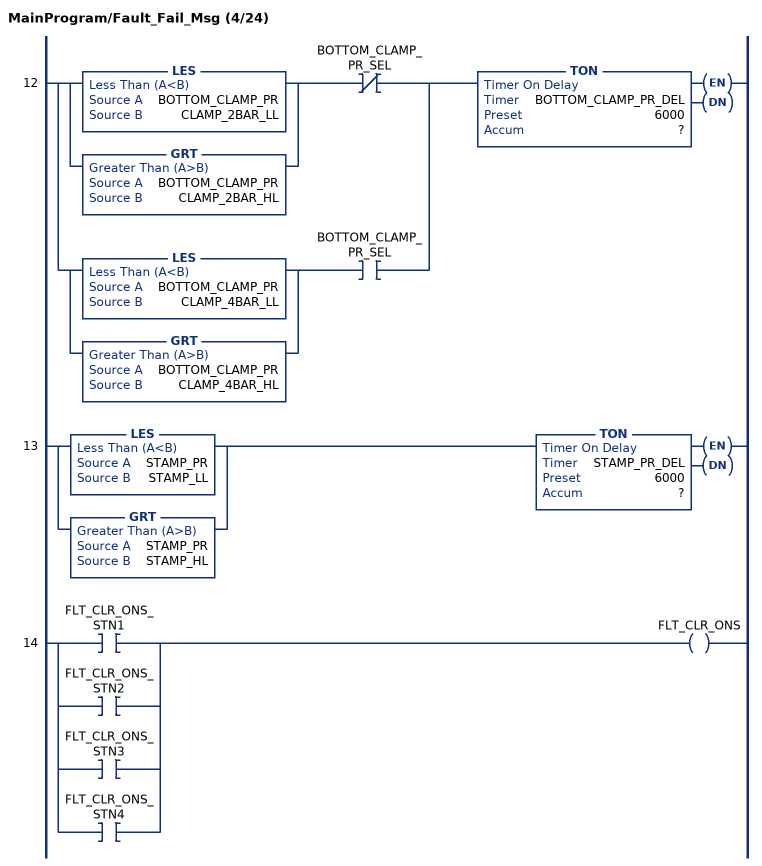
   12: [[LES(BOTTOM_CLAMP_PR,CLAMP_2BAR_LL) ,GRT(BOTTOM_CLAMP_PR,CLAMP_2BAR_HL) ] XIO(BOTTOM_CLAMP_PR_SEL) ,[LES(BOTTOM_CLAMP_PR,CLAMP_4BAR_LL) ,GRT(BOTTOM_CLAMP_PR,CLAMP_4BAR_HL) ] XIC(BOTTOM_CLAMP_PR_SEL) ]TON(BOTTOM_CLAMP_PR_DEL,?,?);
   13: [LES(STAMP_PR,STAMP_LL) ,GRT(STAMP_PR,STAMP_HL) ]TON(STAMP_PR_DEL,?,?);
   14: [XIC(FLT_CLR_ONS_STN1) ,XIC(FLT_CLR_ONS_STN2) ,XIC(FLT_CLR_ONS_STN3) ,XIC(FLT_CLR_ONS_STN4) ]OTE(FLT_CLR_ONS);
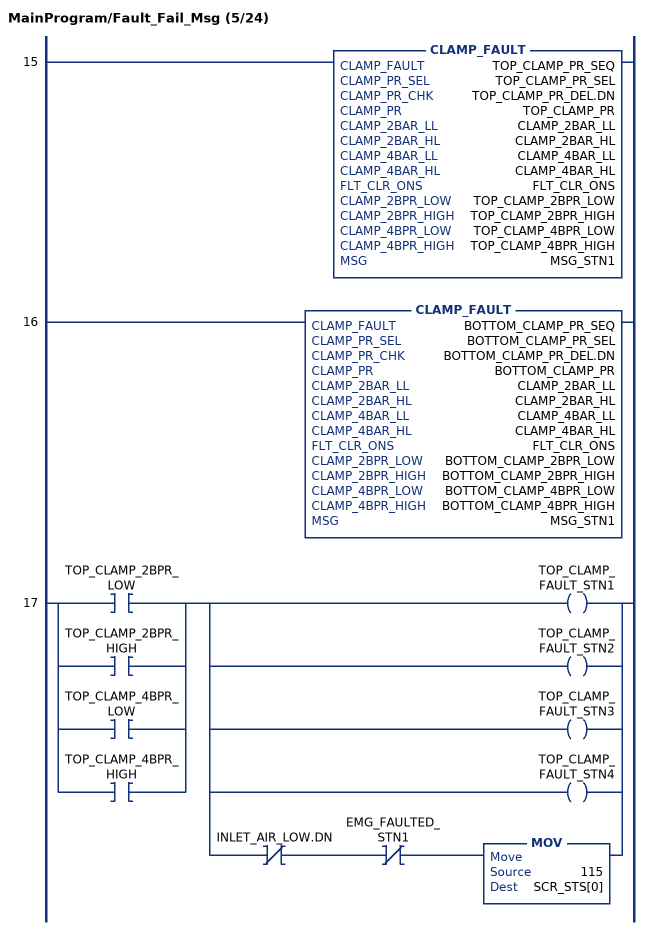
   15: CLAMP_FAULT(TOP_CLAMP_PR_SEQ,TOP_CLAMP_PR_SEL,TOP_CLAMP_PR_DEL.DN,TOP_CLAMP_PR,CLAMP_2BAR_LL,CLAMP_2BAR_HL,CLAMP_4BAR_LL,CLAMP_4BAR_HL,FLT_CLR_ONS,TOP_CLAMP_2BPR_LOW,TOP_CLAMP_2BPR_HIGH,TOP_CLAMP_4BPR_LOW,TOP_CLAMP_4BPR_HIGH,MSG_STN1);
   16: CLAMP_FAULT(BOTTOM_CLAMP_PR_SEQ,BOTTOM_CLAMP_PR_SEL,BOTTOM_CLAMP_PR_DEL.DN,BOTTOM_CLAMP_PR,CLAMP_2BAR_LL,CLAMP_2BAR_HL,CLAMP_4BAR_LL,CLAMP_4BAR_HL,FLT_CLR_ONS,BOTTOM_CLAMP_2BPR_LOW,BOTTOM_CLAMP_2BPR_HIGH,BOTTOM_CLAMP_4BPR_LOW,BOTTOM_CLAMP_4BPR_HIGH,MSG_STN1);
   17: [XIC(TOP_CLAMP_2BPR_LOW) ,XIC(TOP_CLAMP_2BPR_HIGH) ,XIC(TOP_CLAMP_4BPR_LOW) ,XIC(TOP_CLAMP_4BPR_HIGH) ][OTE(TOP_CLAMP_FAULT_STN1) ,OTE(TOP_CLAMP_FAULT_STN2) ,OTE(TOP_CLAMP_FAULT_STN3) ,OTE(TOP_CLAMP_FAULT_STN4) ,XIO(INLET_AIR_LOW.DN) XIO(EMG_FAULTED_STN1) MOV(115,SCR_STS[0]) ];
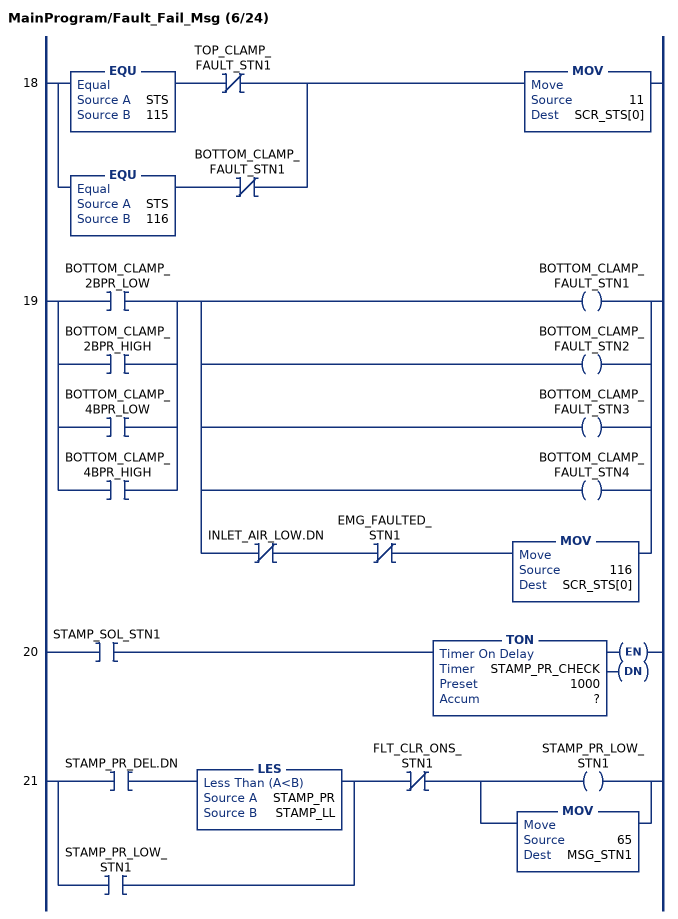
   18: [EQU(STS,115) XIO(TOP_CLAMP_FAULT_STN1) ,EQU(STS,116) XIO(BOTTOM_CLAMP_FAULT_STN1) ]MOV(11,SCR_STS[0]);
   19: [XIC(BOTTOM_CLAMP_2BPR_LOW) ,XIC(BOTTOM_CLAMP_2BPR_HIGH) ,XIC(BOTTOM_CLAMP_4BPR_LOW) ,XIC(BOTTOM_CLAMP_4BPR_HIGH) ][OTE(BOTTOM_CLAMP_FAULT_STN1) ,OTE(BOTTOM_CLAMP_FAULT_STN2) ,OTE(BOTTOM_CLAMP_FAULT_STN3) ,OTE(BOTTOM_CLAMP_FAULT_STN4) ,XIO(INLET_AIR_LOW.DN) XIO(EMG_FAULTED_STN1) MOV(116,SCR_STS[0]) ];
   20: XIC(STAMP_SOL_STN1)TON(STAMP_PR_CHECK,?,?);
   21: [XIC(STAMP_PR_DEL.DN) LES(STAMP_PR,STAMP_LL) ,XIC(STAMP_PR_LOW_STN1) ]XIO(FLT_CLR_ONS_STN1)[OTE(STAMP_PR_LOW_STN1) ,MOV(65,MSG_STN1) ];
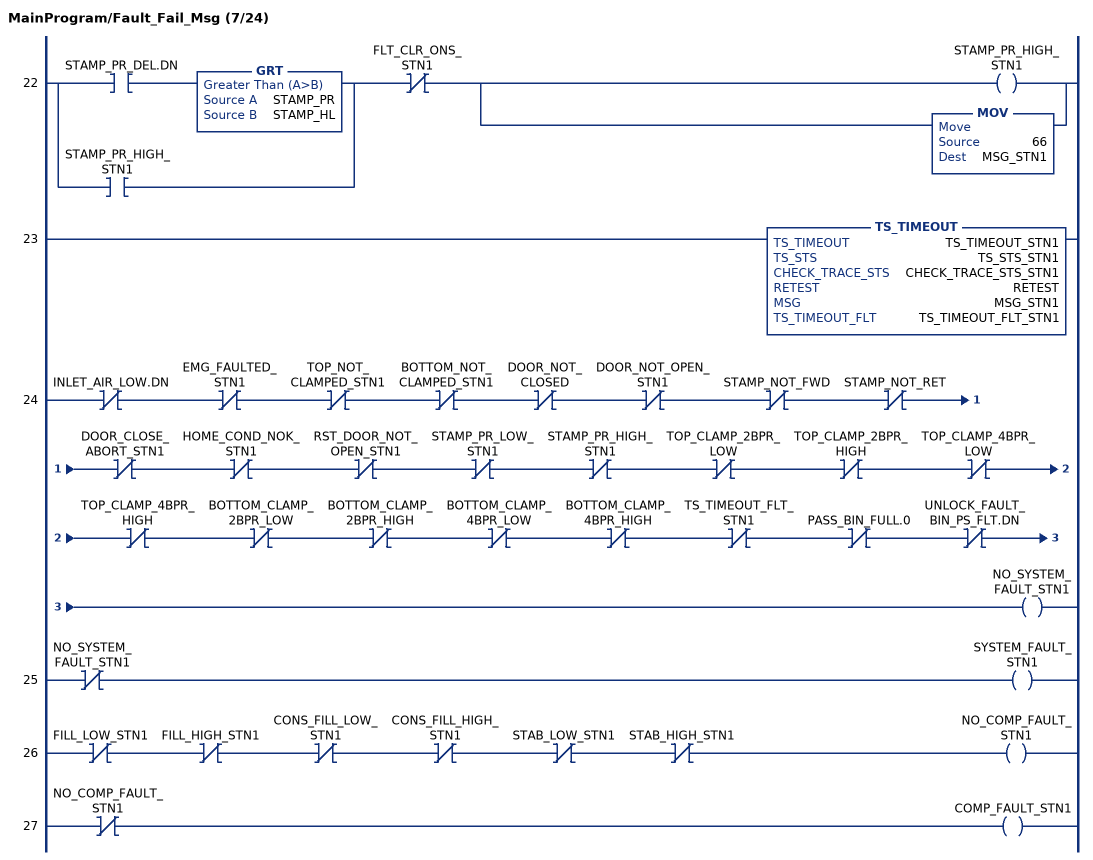
   22: [XIC(STAMP_PR_DEL.DN) GRT(STAMP_PR,STAMP_HL) ,XIC(STAMP_PR_HIGH_STN1) ]XIO(FLT_CLR_ONS_STN1)[OTE(STAMP_PR_HIGH_STN1) ,MOV(66,MSG_STN1) ];
   23: TS_TIMEOUT(TS_TIMEOUT_STN1,TS_STS_STN1,CHECK_TRACE_STS_STN1,RETEST,MSG_STN1,TS_TIMEOUT_FLT_STN1);
   24: XIO(INLET_AIR_LOW.DN)XIO(EMG_FAULTED_STN1)XIO(TOP_NOT_CLAMPED_STN1)XIO(BOTTOM_NOT_CLAMPED_STN1)XIO(DOOR_NOT_CLOSED)XIO(DOOR_NOT_OPEN_STN1)XIO(STAMP_NOT_FWD)XIO(STAMP_NOT_RET)XIO(DOOR_CLOSE_ABORT_STN1)XIO(HOME_COND_NOK_STN1)XIO(RST_DOOR_NOT_OPEN_STN1)XIO(STAMP_PR_LOW_STN1)XIO(STAMP_PR_HIGH_STN1)XIO(TOP_CLAMP_2BPR_LOW)XIO(TOP_CLAMP_2BPR_HIGH)XIO(TOP_CLAMP_4BPR_LOW)XIO(TOP_CLAMP_4BPR_HIGH)XIO(BOTTOM_CLAMP_2BPR_LOW)XIO(BOTTOM_CLAMP_2BPR_HIGH)XIO(BOTTOM_CLAMP_4BPR_LOW)XIO(BOTTOM_CLAMP_4BPR_HIGH)XIO(TS_TIMEOUT_FLT_STN1)XIO(PASS_BIN_FULL.0)XIO(UNLOCK_FAULT_BIN_PS_FLT.DN)OTE(NO_SYSTEM_FAULT_STN1);
   25: XIO(NO_SYSTEM_FAULT_STN1)OTE(SYSTEM_FAULT_STN1);
   26: XIO(FILL_LOW_STN1)XIO(FILL_HIGH_STN1)XIO(CONS_FILL_LOW_STN1)XIO(CONS_FILL_HIGH_STN1)XIO(STAB_LOW_STN1)XIO(STAB_HIGH_STN1)OTE(NO_COMP_FAULT_STN1);
   27: XIO(NO_COMP_FAULT_STN1)OTE(COMP_FAULT_STN1);
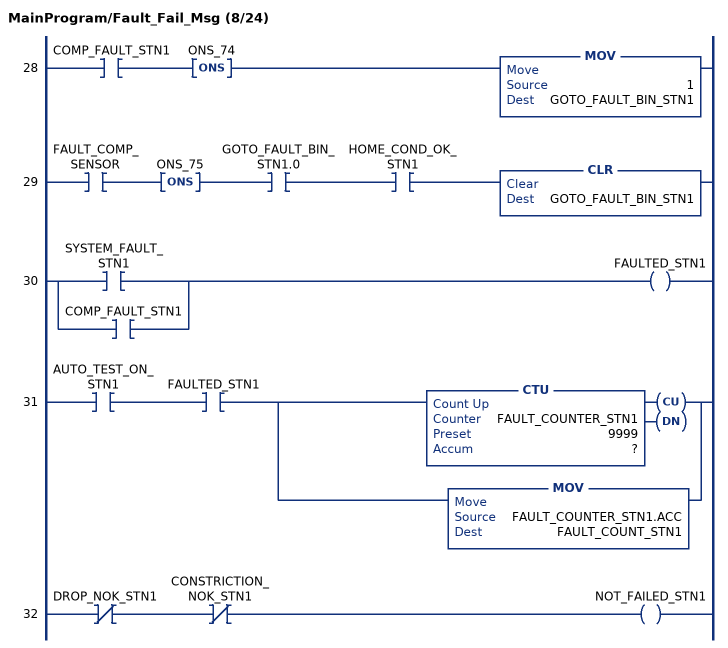
   28: XIC(COMP_FAULT_STN1)ONS(ONS_74)MOV(1,GOTO_FAULT_BIN_STN1);
   29: XIC(FAULT_COMP_SENSOR)ONS(ONS_75)XIC(GOTO_FAULT_BIN_STN1.0)XIC(HOME_COND_OK_STN1)CLR(GOTO_FAULT_BIN_STN1);
   30: [XIC(SYSTEM_FAULT_STN1) ,XIC(COMP_FAULT_STN1) ]OTE(FAULTED_STN1);
   31: XIC(AUTO_TEST_ON_STN1)XIC(FAULTED_STN1)[CTU(FAULT_COUNTER_STN1,?,?) ,MOV(FAULT_COUNTER_STN1.ACC,FAULT_COUNT_STN1) ];
   32: XIO(DROP_NOK_STN1)XIO(CONSTRICTION_NOK_STN1)OTE(NOT_FAILED_STN1);
